// TIA Portal V19 export
DATA_BLOCK "Lubr_Bordat_DB"   // DB227
// stored: InstanceOfName Lubr_Bordat, InstanceOfType FB
"Lubr_Bordat"
   // VAR
   //    Ton_Stop : TON_TIME;
   //    Ton_Start : TON_TIME;
   //    Ctrl { S7_SetPoint := 'True'} : Bool;
   //    Abilita : Bool;
   // END_VAR
BEGIN
END_DATA_BLOCK
